// TIA Portal project "bb2-G1" (V14)

(* hardware
DEVICE "S7-1200 station_1"  S7-1200 Station
   slot 0: "Rack_0"  Rack  V1.0
   slot 1: "PLC_1"  CPU 1214C DC/DC/DC  6ES7 214-1AG40-0XB0  V4.0
*)

// ===== PLC "PLC_1"  CPU 1214C DC/DC/DC =====

VAR_GLOBAL   // PLC tag table "Default tag table"
   "Axis_1_Homing switch" AT %I0.0 : Bool;
   "Axis_1_LowHwLimitSwitch" AT %I0.6 : Bool;
   "Axis_1_HighHwLimitSwitch" AT %I0.7 : Bool;
   "Axis_1_Homing switch(1)" AT %I0.5 : Bool;
   "Axis_1_Pulse" AT %Q0.0 : Bool;
   "Axis_1_Direction" AT %Q0.2 : Bool;
   "Axis_1_DriveEnable" AT %Q0.3 : Bool;
   "Tag_1" AT %Q0.5 : Bool;
   "Tag_2" AT %Q0.4 : Bool;
   "Tag_3" AT %I0.4 : Bool;
   "Tag_4" AT %I0.2 : Bool;
   "Tag_5" AT %I0.1 : Bool;
   "Tag_6" AT %MD33 : Real;
   "Tag_7" AT %I0.3 : Bool;
END_VAR

DATA_BLOCK "Axis_1"   // DB1, Motion_DB
{ S7_Optimized_Access := 'TRUE' }
AUTHOR : SIMATIC
FAMILY : BasicMC
NAME : TO_PosAx
VERSION : 4.0
// stored: InstanceOfName TO_PositioningAxis
"TO_PositioningAxis"
BEGIN
   // Axis.PositionLimitsMax_AddressCU = %I0.7
   // Axis.PositionLimitsMin_AddressCU = %I0.6
   // Axis.LengthUnit.LastDistance = 1005
   // Axis.HomingReferencePointSwitch_AddressCU = %I0.5
   // Axis.DirectionOutputEnabledCU = TRUE
   // Axis.OnlinePtoModeCUEnumValue = PTO (pulse A and direction B)
   // Axis.OnlinePtoModeCU = 16#0000_0002
   // Axis.SelectedChannel2EnumCU = %Q0.2
   // Axis.SelectedChannel1EnumCU = %Q0.0
   // Pulse.MinDeltaDeltaFrequencyCU = 0.004
   // Pulse.MaxDeltaDeltaFrequencyCU = 1.0E+10
   // Pulse.MinDeltaFrequencyCU = 0.005
   // Pulse.MaxDeltaFrequencyCU = 9.5E+9
   // Pulse.MinFrequencyCU = 1.0
   // Pulse.MaxFrequencyCU = 100000.0
   // Pulse.OutputSourceCU = 16#0000_0000
   // Axis.SelectPTO = 0
END_DATA_BLOCK

ORGANIZATION_BLOCK "Main"   // OB1, LAD, ProgramCycle
TITLE = "Main Program Sweep (Cycle)"
{ S7_Optimized_Access := 'TRUE' }
VERSION : 0.1
   VAR_INPUT
      Initial_Call : Bool;   // Initial call of this OB
      Remanence : Bool;   // =True, if remanent data are available
   END_VAR
BEGIN

REGION Network 1
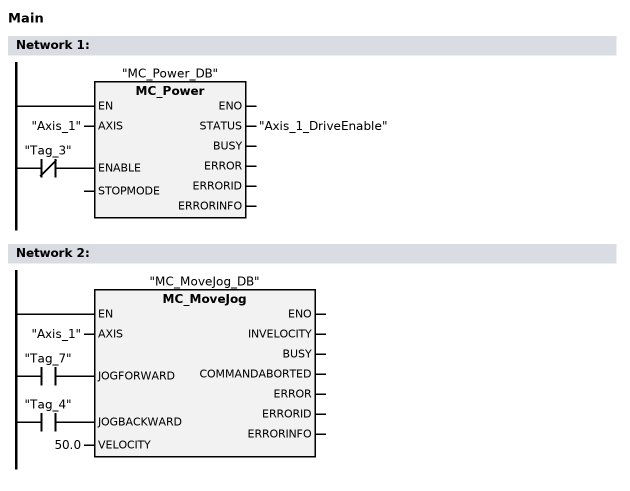
   "MC_Power_DB"(Axis := "Axis_1", Enable := NOT "Tag_3", Status => "Axis_1_DriveEnable");   // MC_Power
END_REGION

REGION Network 2
   "MC_MoveJog_DB"(Axis := "Axis_1", JogForward := "Tag_7", JogBackward := "Tag_4", Velocity := 50.0);   // MC_MoveJog
END_REGION
END_ORGANIZATION_BLOCK